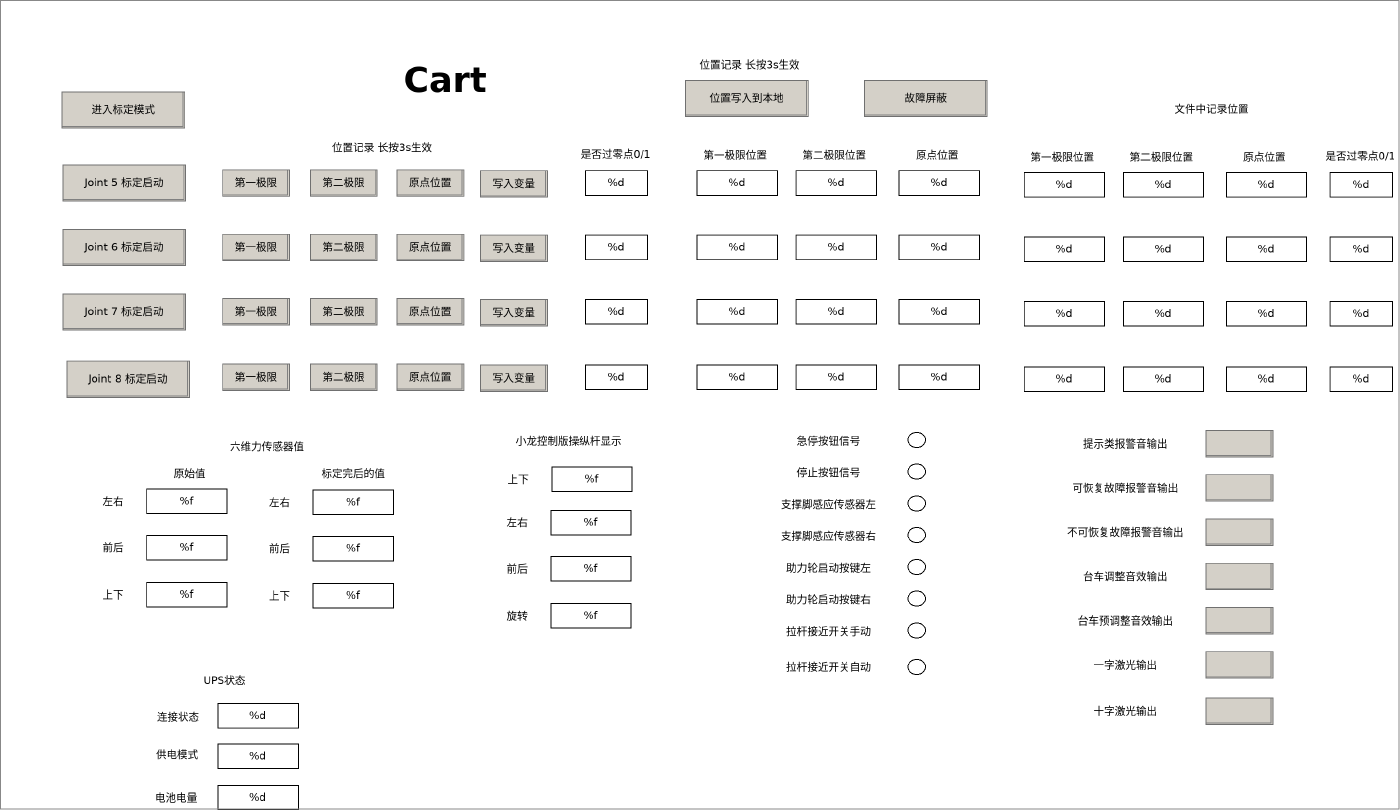
VISUALIZATION carCail  // 1455x842
    Button (64,95 128x38), "进入标定模式", colour toggle: GVL_armCali.g_CartEnterCaliMode
        toggle GVL_armCali.g_CartEnterCaliMode
    Button (65,171 128x38), "Joint 5 标定启动", colour toggle: GVL_armCali.g_jointIntoCaliStateOfCart[5]
        tap GVL_armCali.g_jointIntoCaliStateOfCart[5]
    Button (231,176 70x28), "第一极限", colour toggle: GVL_armCali.g_linkEncFristCaliTriggerOfCart[5]
        tap GVL_armCali.g_linkEncFristPosCaliOfCart[5]
    Button (322,176 70x28), "第二极限", colour toggle: GVL_armCali.g_linkEncSecondCaliTriggerOfCart[5]
        tap GVL_armCali.g_linkEncSecondPosCaliOfCart[5]
    Rectangle (608,177 65x26), "%d", text variable: GVL_armCali.g_linkZeroCrossOrNotOfCart[5]
    Rectangle (724,177 84x26), "%d", text variable: GVL_armCali.g_linkLimitFristPosOfCart[5]
    Rectangle (827,177 84x26), "%d", text variable: GVL_armCali.g_linkLimitSecondPosOfCart[5]
    Rectangle (934,177 84x26), "%d", text variable: GVL_armCali.g_linkHomePosOfCart[5]
    Button (412,176 70x28), "原点位置", colour toggle: GVL_armCali.g_linkEncHomePosCaliTriggerOfCart[5]
        tap GVL_armCali.g_linkEncHomePosCaliOfCart[5]
    Button (65,238 128x38), "Joint 6 标定启动", colour toggle: GVL_armCali.g_jointIntoCaliStateOfCart[6]
        tap GVL_armCali.g_jointIntoCaliStateOfCart[6]
    Button (231,243 70x28), "第一极限", colour toggle: GVL_armCali.g_linkEncFristCaliTriggerOfCart[6]
        tap GVL_armCali.g_linkEncFristPosCaliOfCart[6]
    Button (322,243 70x28), "第二极限", colour toggle: GVL_armCali.g_linkEncSecondCaliTriggerOfCart[6]
        tap GVL_armCali.g_linkEncSecondPosCaliOfCart[6]
    Rectangle (608,244 65x26), "%d", text variable: GVL_armCali.g_linkZeroCrossOrNotOfCart[6]
    Rectangle (724,244 84x26), "%d", text variable: GVL_armCali.g_linkLimitFristPosOfCart[6]
    Rectangle (827,244 84x26), "%d", text variable: GVL_armCali.g_linkLimitSecondPosOfCart[6]
    Rectangle (934,244 84x26), "%d", text variable: GVL_armCali.g_linkHomePosOfCart[6]
    Button (412,243 70x28), "原点位置", colour toggle: GVL_armCali.g_linkEncHomePosCaliTriggerOfCart[6]
        tap GVL_armCali.g_linkEncHomePosCaliOfCart[6]
    Button (65,305 128x38), "Joint 7 标定启动", colour toggle: GVL_armCali.g_jointIntoCaliStateOfCart[7]
        tap GVL_armCali.g_jointIntoCaliStateOfCart[7]
    Button (231,310 70x28), "第一极限", colour toggle: GVL_armCali.g_linkEncFristCaliTriggerOfCart[7]
        tap GVL_armCali.g_linkEncFristPosCaliOfCart[7]
    Button (322,310 70x28), "第二极限", colour toggle: GVL_armCali.g_linkEncSecondCaliTriggerOfCart[7]
        tap GVL_armCali.g_linkEncSecondPosCaliOfCart[7]
    Rectangle (608,311 65x26), "%d", text variable: GVL_armCali.g_linkZeroCrossOrNotOfCart[7]
    Rectangle (724,311 84x26), "%d", text variable: GVL_armCali.g_linkLimitFristPosOfCart[7]
    Rectangle (827,311 84x26), "%d", text variable: GVL_armCali.g_linkLimitSecondPosOfCart[7]
    Rectangle (934,311 84x26), "%d", text variable: GVL_armCali.g_linkHomePosOfCart[7]
    Button (412,310 70x28), "原点位置", colour toggle: GVL_armCali.g_linkEncHomePosCaliTriggerOfCart[7]
        tap GVL_armCali.g_linkEncHomePosCaliOfCart[7]
    Button (69,375 128x38), "Joint 8 标定启动", colour toggle: GVL_armCali.g_jointIntoCaliStateOfCart[8]
        tap GVL_armCali.g_jointIntoCaliStateOfCart[8]
    Button (231,378 70x28), "第一极限", colour toggle: GVL_armCali.g_linkEncFristCaliTriggerOfCart[8]
        tap GVL_armCali.g_linkEncFristPosCaliOfCart[8]
    Button (322,378 70x28), "第二极限", colour toggle: GVL_armCali.g_linkEncSecondCaliTriggerOfCart[8]
        tap GVL_armCali.g_linkEncSecondPosCaliOfCart[8]
    Rectangle (608,379 65x26), "%d", text variable: GVL_armCali.g_linkZeroCrossOrNotOfCart[8]
    Rectangle (724,379 84x26), "%d", text variable: GVL_armCali.g_linkLimitFristPosOfCart[8]
    Rectangle (827,379 84x26), "%d", text variable: GVL_armCali.g_linkLimitSecondPosOfCart[8]
    Rectangle (934,379 84x26), "%d", text variable: GVL_armCali.g_linkHomePosOfCart[8]
    Button (412,378 70x28), "原点位置", colour toggle: GVL_armCali.g_linkEncHomePosCaliTriggerOfCart[8]
        tap GVL_armCali.g_linkEncHomePosCaliOfCart[8]
    Rectangle (1064,179 84x26), "%d", text variable: GVL_CartJointEncoderCaliData.g_minLinkEncoder[5]
    Rectangle (1167,179 84x26), "%d", text variable: GVL_CartJointEncoderCaliData.g_maxLinkEncoder[5]
    Rectangle (1274,179 84x26), "%d", text variable: GVL_CartJointEncoderCaliData.g_caliLinkEncoder[5]
    Rectangle (1064,246 84x26), "%d", text variable: GVL_CartJointEncoderCaliData.g_minLinkEncoder[6]
    Rectangle (1167,246 84x26), "%d", text variable: GVL_CartJointEncoderCaliData.g_maxLinkEncoder[6]
    Rectangle (1274,246 84x26), "%d", text variable: GVL_CartJointEncoderCaliData.g_caliLinkEncoder[6]
    Rectangle (1064,313 84x26), "%d", text variable: GVL_CartJointEncoderCaliData.g_minLinkEncoder[7]
    Rectangle (1167,313 84x26), "%d", text variable: GVL_CartJointEncoderCaliData.g_maxLinkEncoder[7]
    Rectangle (1274,313 84x26), "%d", text variable: GVL_CartJointEncoderCaliData.g_caliLinkEncoder[7]
    Rectangle (1064,381 84x26), "%d", text variable: GVL_CartJointEncoderCaliData.g_minLinkEncoder[8]
    Rectangle (1167,381 84x26), "%d", text variable: GVL_CartJointEncoderCaliData.g_maxLinkEncoder[8]
    Rectangle (1274,381 84x26), "%d", text variable: GVL_CartJointEncoderCaliData.g_caliLinkEncoder[8]
    Rectangle (1382,179 65x26), "%d", text variable: GVL_CartJointEncoderCaliData.g_linkEncZeroCross[5]
    Rectangle (1382,246 65x26), "%d", text variable: GVL_CartJointEncoderCaliData.g_linkEncZeroCross[6]
    Rectangle (1382,313 65x26), "%d", text variable: GVL_CartJointEncoderCaliData.g_linkEncZeroCross[7]
    Rectangle (1382,381 65x26), "%d", text variable: GVL_CartJointEncoderCaliData.g_linkEncZeroCross[8]
    Button (499,177 70x28), "写入变量", colour toggle: GVL_armCali.g_linkPosWriteCaliDataTriggerOfCart[5]
        tap GVL_armCali.g_linkPosWriteCaliDataOfCart[5]
    Button (499,244 70x28), "写入变量", colour toggle: GVL_armCali.g_linkPosWriteCaliDataTriggerOfCart[6]
        tap GVL_armCali.g_linkPosWriteCaliDataOfCart[6]
    Button (499,311 70x28), "写入变量", colour toggle: GVL_armCali.g_linkPosWriteCaliDataTriggerOfCart[7]
        tap GVL_armCali.g_linkPosWriteCaliDataOfCart[7]
    Button (499,379 70x28), "写入变量", colour toggle: GVL_armCali.g_linkPosWriteCaliDataTriggerOfCart[8]
        tap GVL_armCali.g_linkPosWriteCaliDataOfCart[8]
    Label (599,149 82x23), "是否过零点0/1"
    Label (364,57 197x52), "Cart"
    Label (723,150 82x23), "第一极限位置"
    Label (826,150 82x23), "第二极限位置"
    Label (322,142 150x23), "位置记录 长按3s生效"
    Label (933,150 82x23), "原点位置"
    Button (712,83 128x38), "位置写入到本地", colour toggle: GVL_armCali.g_caliDataWriteTriggerOfCart
        tap GVL_armCali.g_caliDataWriteOfCart
    Label (704,56 150x23), "位置记录 长按3s生效"
    Label (1063,152 82x23), "第一极限位置"
    Label (1166,152 82x23), "第二极限位置"
    Label (1273,152 82x23), "原点位置"
    Label (1184,102 150x23), "文件中记录位置"
    Label (1373,151 82x23), "是否过零点0/1"
    Button (898,83 128x38), "故障屏蔽", colour toggle: g_specialSignal.m_faultMask[1]
        toggle g_specialSignal.m_faultMask[1]
    Rectangle (152,508 84x26), "%f", text variable: GVL_IO.g_sixForceOrigin[1]
    Label (219,453 117x23), "六维力传感器值"
    Label (91,510 53x23), "左右"
    Label (162,481 70x23), "原始值"
    Rectangle (152,556 84x26), "%f", text variable: GVL_IO.g_sixForceOrigin[2]
    Label (91,558 53x23), "前后"
    Rectangle (152,605 84x26), "%f", text variable: GVL_IO.g_sixForceOrigin[3]
    Label (91,607 53x23), "上下"
    Rectangle (325,509 84x26), "%f", text variable: GVL_IO.g_sixForceCali[1]
    Label (264,511 53x23), "左右"
    Label (319,481 96x23), "标定完后的值"
    Rectangle (325,557 84x26), "%f", text variable: GVL_IO.g_sixForceCali[2]
    Label (264,559 53x23), "前后"
    Rectangle (325,606 84x26), "%f", text variable: GVL_IO.g_sixForceCali[3]
    Label (264,608 53x23), "上下"
    Label (501,447 180x23), "小龙控制版操纵杆显示"
    Rectangle (572,530 84x26), "%f", text variable: GVL_IO.g_joystickSignalAnalysis[2]
    Label (511,532 53x23), "左右"
    Rectangle (572,578 84x26), "%f", text variable: GVL_IO.g_joystickSignalAnalysis[3]
    Label (511,580 53x23), "前后"
    Rectangle (572,627 84x26), "%f", text variable: GVL_IO.g_joystickSignalAnalysis[4]
    Label (511,629 53x23), "旋转"
    Rectangle (573,485 84x26), "%f", text variable: GVL_IO.g_joystickSignalAnalysis[1]
    Label (512,487 53x23), "上下"
    Label (821,447 80x23), "急停按钮信号"
    Ellipse (943,449 19x16), colour toggle: GVL_IO.g_emergencyStopButton
    Label (821,480 80x23), "停止按钮信号"
    Ellipse (943,482 19x16), colour toggle: GVL_IO.g_stopButton
    Label (791,513 140x23), "支撑脚感应传感器左"
    Ellipse (943,515 19x16), colour toggle: GVL_IO.g_supportLegSensor[1]
    Label (791,546 140x23), "支撑脚感应传感器右"
    Ellipse (943,548 19x16), colour toggle: GVL_IO.g_supportLegSensor[2]
    Label (791,579 140x23), "助力轮启动按键左"
    Ellipse (943,581 19x16), colour toggle: GVL_IO.g_carHandChassisDriveUnlock[1]
    Label (791,612 140x23), "助力轮启动按键右"
    Ellipse (943,614 19x16), colour toggle: GVL_IO.g_carHandChassisDriveUnlock[2]
    Label (791,645 140x23), "拉杆接近开关手动"
    Ellipse (943,647 19x16), colour toggle: GVL_IO.g_drivingLeverSensor[1]
    Label (791,682 140x23), "拉杆接近开关自动"
    Ellipse (943,685 19x16), colour toggle: GVL_IO.g_drivingLeverSensor[2]
    Button (1253,447 70x28), colour toggle: GVL_IO.g_openWarningTone[1]
        tap GVL_IO.g_openWarningTone[1]
    Label (1109,450 121x23), "提示类报警音输出"
    Button (1253,493 70x28), colour toggle: GVL_IO.g_openWarningTone[2]
        tap GVL_IO.g_openWarningTone[2]
    Label (1100,496 139x23), "可恢复故障报警音输出"
    Button (1253,539 70x28), colour toggle: GVL_IO.g_openWarningTone[3]
        tap GVL_IO.g_openWarningTone[3]
    Label (1095,542 149x23), "不可恢复故障报警音输出"
    Button (1253,585 70x28), colour toggle: GVL_IO.g_openWarningTone[4]
        tap GVL_IO.g_openWarningTone[4]
    Label (1095,588 149x23), "台车调整音效输出"
    Button (1253,631 70x28), colour toggle: GVL_IO.g_openWarningTone[5]
        tap GVL_IO.g_openWarningTone[5]
    Label (1095,634 149x23), "台车预调整音效输出"
    Button (1253,677 70x28), colour toggle: GVL_IO.g_openHorizonLaser
        tap GVL_IO.g_openHorizonLaser
    Label (1095,680 149x23), "一字激光输出"
    Button (1253,725 70x28), colour toggle: GVL_IO.g_openCrossLaser
        tap GVL_IO.g_openCrossLaser
    Label (1095,728 149x23), "十字激光输出"
    Label (197,696 73x23), "UPS状态"
    Rectangle (226,816 84x26), "%d", text variable: GVL_interactUI.g_dumpEnergyUPS
    Label (148,818 70x23), "电池电量"
    Label (149,773 70x23), "供电模式"
    Label (150,734 70x23), "连接状态"
    Rectangle (226,773 84x26), "%d", text variable: GVL_interactUI.g_powerSupplyModeUPS
    Rectangle (226,731 84x26), "%d", text variable: GVL_interactUI.g_upsComStatus
END_VISUALIZATION

(* stored: Version 1.1.0.1, ProductVersion 3.1.4024.11
   Visu carCail: Id {761fe35a-e76f-46c0-8e2a-58082bc85c4b} *)
